# B&R Automation Studio project dbserv_0640 (part 13)

#### iec60870_5_103.c
```c
#ifdef _DEFAULT_INCLUDES
	#include <AsDefault.h>
#endif
/******************************************************************************
*    COPYRIGHT    BERNECKER + RAINER Industrie-Elektronik Ges.m.b.H           *
*******************************************************************************
*  Projekt:  Protokoll Treiber IEC 60870-5-103
*  Teil:     Hauptprogramm
*  Datei:    iec60870_5_103.c
*  Typ:      GNU-C (32 Bit)
*------------------------------------------------------------------------------
*  Revision: 03.00.5
*  Datum:    07-02-2019
*  Autor:    KOB
*------------------------------------------------------------------------------
*  Funktion:
*------------------------------------------------------------------------------
*  Rev.   | Datum    | Name | Kommentar
*  -------+----------+------+---------------------------------------------------
*  01.00  | 26-11-03 | KOB  | Datei-Erstellung
*  01.01  | 09-02-04 | KOB  | Debugkonfiguration um Liniennummer erweitert
*         |          |      | Meldung an LS, falls Schnittstelle nicht geöffnet werden
*		  |          |      | kann, dabei warten bis myidBrServer!= 0 ist.
*  01.02  | 07-05-04 | KOB  | Verbindungsstoerung bei Initialisierung auf 1 setzen, damit
*		  |          |      | beim ersten gültigen Telegramm der Datenpunkt Kopplungsstoerung
*		  |          |      | beschrieben wird.
*  01.03  | 15-12-04 | KOB  | Bei ungültigen Analogwerten (Invalid oder Overflow) wird
*         |          |      | als Ersatzwert 7FFF gesendet.
*  01.04  | 11-04-06 | WAI  | FileIO-Library includiert wegen neuer dbServ-Version mit Archivierung
*  01.05  | 24-05-06 | KOB  | Telegrammauswertung flexibler gestaltet (wegen anderem Verhalten von ABB)
*		  |          |      |
*  01.06  | 10-01-07 | KOB  | Erweiterung um die Telegramme:
*         |          |      | Type Identification 3 : Measurands 1
*         |          |      | (check_m3, iec__103_sub.c)
*         |          |      | Type Identification 79: Privates Telegramm zur Übertragung von Zählwerten
*         |          |      | (check_m79, iec__103_sub.c)
*         |          |      | Auswertung der im privaten Telegramm empfangenen Zählwerte
*         |          |      | (save_analogwert_priv, iec__103_serv.c)
*		  |          |      |
*  02.05.1| 02-09-08 | KOB  | Neue Modi für Doppelmeldungen:
*		  |			 |		| DOPPEL_EINZEL_NORMAL_NOINVALID und DOPPEL_EINZEL_INVERS_NOINVALID
*		  |          |      |
*		  |			 |		| KE_Init: Bei der Auswertungt des Rückmeldetelegrammes
*		  |			 |		| Identification Message (check_m5) wird die Überprüfung des
*		  |			 |		| Function Type weggelassen, d.h. es wird für alle Geräte aktzeptiert.
*		  |			 |		| Bisher wurde das Telegramm nur für Function Type 160,192,240 zugelassen.
*		  |          |      |
*         |          |      |
*  02.05.2| 02-09-08 | KOB  | Funktionen wie unter 01.06 beschrieben eingefügt.
*         |          |      |
*  02.06.4| 27-09-10 | WAI  | IsANumber() mit Vorzeichen
*         |          |      |
*  02.07.2| 26-07-11 | KOB  | Erweiterung um die Telegramme:
*         |          |      | Type Identification 205: Privates Telegramm zur Übertragung von Zählwerten (Siemens)
*         |          |      | (check_m205, iec__103_sub.c)
*         |          |      | Auswertung der im privaten Telegramm empfangenen Zählwerte
*         |          |      | (save_counter_2, iec__103_serv.c)
*         |          |      |
* 		  |			 | KOB  | Ueberwachung der Zeitsynchronisation:
*         |          |      | Parameter IEC Global: Timeout fuer Rueckmeldung Zeitsyncronisation (TIME.TIMEOUT)
*         |          |      | Parameter pro Gerät : ERR.TIMESYNC
*  02.07.3| 04-12-13 | KOB  | check_m5 angepasst: Zustand von ACD Bit ignoriert, Kompatibilitätsmodus 3 akzeptieren
*         |          |      | check_m6 angepasst: nicht verwendete Bits der zurueckgemeldeten Zeit ausmaskieren
*         |          |      | neue Debug Möglichkeit (Variablen: IEC_Info_Clear,IEC_Info_Enable,IEC_InfoNumber,IEC_Info)
*         |          |      | Aufschlüsselung der IEC Telegrammsteuerelemente und Eintrag in Buffer
*  03.00.2| 28-01-14 | KOB  | check_m5 angepasst: Info Nr 2 akzeptieren
*         |          |      | Defaultwert für IEC_Config.TimeClass2PollFast von 100ms auf 200ms erhöht
*  03.00.3| 04-04-14 | KOB  | TIME_DIFF_SYNCH_MAX von 2 auf 10 geändert
*         |          |      | DeviceActivType erweitert um die Elemente
*         |          |      | TDiff und TDiffCounter;
*         |          |      | check_m6() Uhrzeitdifferenz wird in Struktur eingetragen
*         |          |      | Ist die Uhrzeitdifferenz zu groß, wird erste beim 2.Mal Felhler generiert
*  03.00.4| 11-10-16 | WAI  | Änderungen tbd (BIE)
*  03.00.5| 07-02-19 | KOB  | Senden von Kommandos überarbeitet

******************************************************************************/

/***********************************************************************/
/* Headerfiles einbinden                                               */
/***********************************************************************/

#include <bur\plc.h>			/* RPS-spezifische Typendeklarationen */
#include <string.h>
#include <dvframe.h>
#include <asbrstr.h>
#include <sys_lib.h>
#include <brsystem.h>
#include <fileio.h>
#include "iec__103_date.h"		/* Funktionen zur Datumsberechnung */
#include "iec60870_5_103.h"		/* Definition der globalen Variablen */
#include "iec__103_debug.h"		/* Funktionen fuer Ausgabe von Debug-Meldungen */
#include "iec__103_parse.h"		/* Parser Funktionen */
#include "dbserv.h"				/* Meldeserver */

extern DebugConfig_typ	DebugConfig;

/***********************************************************************/
/* 					Initialisierungs-Unterprogramm                     */
/***********************************************************************/

void _INIT init_iec(void)
{
	signed short i,n;

	/*--------------------------------*/
	/* Variablen initialisieren       */
	/*--------------------------------*/
	for(i=0;i<ITEM_DIAGNOSE_SIZE;i++) {
		IEC_ItemDiagnose[i].showData	= 0;
	}
	IEC_NormDiagnose.showData			= 0;

	dbg_buf_iec_clear();
	IEC_Info_Clear	= 0;
	IEC_Info_Enable = 0;

	memset(&SYS_Statistic,0,sizeof(SYS_Statistic));
	memset(&DistDataServer,0,sizeof(DistDataServer));						/* Variable fuer die Uebergabe von Stoerschrieben an das Leitsystem */
	memset(&stANL,0,sizeof(stANL));											/* Variable für Linien und Geräteverwaltung */
	memset(&stComIni,0,sizeof(stComIni));									/* Variable zur Verwaltung der Schnittstellen */

	myidBrServer			= 0;											/* ID BR-Server */
	DisturbanceSimulation	= 0;											/* Merker zur Simulation eines Stoerschriebes */

	rt_info.enable = 1; 													/* Taskklassenzykluszeit ermitteln */
	RTInfo(&rt_info);
	if(rt_info.status==0)	CycleTime	= (rt_info.cycle_time / 1000);		/* Zykluszeit in ms */
	else 					CycleTime	= 10;								/* Zykluszeit in ms */

	DebugConfig.OpenDevice			= 0;									/* Debug Funktion deaktivieren */
	DebugConfig.DebugEnable			= 0;
	DebugConfig.DebugDelayAdresse	= 0;
	DebugConfig.DebugDelayTime		= 0;
	DebugConfig.DebugDelayCounter	= 0;

	Error	= 0;															/* Generelle Variable fuer Initialisierungsfehler */

	/*----------------------------------------------------------------------*/
	/* initialize debugging 												*/
	/*----------------------------------------------------------------------*/

	#ifdef DEBUG
		debug_initialize();
	#endif

	/*--------------------------------------------------*/
	/* Globale Konfigurationsparameter initialisieren	*/
	/*--------------------------------------------------*/

	IEC_Config.TimeOut				= 100;				/* Timeout bei Telegrammempfang (in ms) */
	IEC_Config.RetryAnz				= 6;				/* Anzahl Telegrammwiederholungen bei bestehender Verbindung */
	IEC_Config.ConnAnz				= 3;				/* Anzahl Telegrammwiederholung bei neu aufzubauender Verbindung */
	IEC_Config.WaitIntv				= 100000;			/* Wartezeit für erneuten Verbindungsaufbau (in ms) */
	IEC_Config.TimeTS				= 60000;			/* Intervallzeit fuer Uhrzeitsynchronisation (in ms) */
	IEC_Config.TimeOutTimeSynch		= 10000;			/* Timeout fuer die Rückantwort bei Zeitsynchronisation in (ms) */
	IEC_Config.EnableComReset		= 1;				/* Freigabe fuer das Schliessen und Wieder-Oeffnen der Schnittstelle bei Schreibfehlern */
	IEC_Config.TimeClass2Poll		= 1000;				/* Abtastzeit Class 2 Telegramme (Analogwerte) (in ms) */
	IEC_Config.TimeClass2PollFast	= 200;				/* Abtastzeit Class 2 Telegramme (Analogwerte) (in ms) während Übertragung von Störschrieben in ms */
	IEC_Config.DistDataTimeoutMax	= 20000;			/* Timeout fuer den Telegrammempfang bei Stoerschriebuebertragung in (ms) */
	IEC_Config.DistDataEnable		= 1;				/* Freigabe fuer Stoerschriebuebertragung */
	IEC_Config.DisturbanceDelay		= 10000;			/* Zeit die ein Lesen von Stoerschrieben der gleichen Station verzoegert wird in (ms) */
	IEC_Config.CommandEnable		= 0;				/* Freigabe für die Übertragung von Kommandos */
	IEC_Config.CommandTimeoutMax	= 40000;			/* Timeout fuer die Uebertragung von Kommandos in (ms) */

	/*****************************************************************************/
	/* Initialisierung nach Konfigurationsdatenmodul dplist und typlist (DbServ) */
	/*****************************************************************************/
#ifdef INIT_MODE_DM_DPLIST

	/*--------------------------------------------------*/
	/* Konfiguration aus Konfigurationsmodulen auslesen */
	/*--------------------------------------------------*/

	for(aktANL= 0; aktANL < MAX_LINES; aktANL++) {
		for(n = 0; n < DEVICES_PRO_LINE; n++) {
			stANL[aktANL].DeviceActiv[n].FaultFunctionType		= 160; /* Vorbelegung, wird später vom Telegramm des Geräts übernommen */
		}
	}

	iec_parser();

	Error = IEC_ParserInfo.error;

	/* Kein Schwerwiegender Fehler beim Parsen */
	if(Error==0) {
		/* Maximale Anzahl Linien (Endevariable für Schleifen) */
		if(IEC_ParserInfo.NrOfLines>0) {
			maxANL = IEC_ParserInfo.NrOfLines - 1;
		}
		else {
			maxANL = 0;
		}

		for(aktANL= 0; aktANL <= maxANL; aktANL++) {
			stANL[aktANL].LinienNummer			= IEC_GlobalData.Line[aktANL].LineNr.value;
			stANL[aktANL].Error					= IEC_ParserInfo.Line[aktANL].error;
			stANL[aktANL].dm.AdrDM_norm			= IEC_ParserInfo.memAdr;
			stANL[aktANL].dm.MaxWerteDM_norm	= IEC_ParserInfo.NrOfNormValues;
			stANL[aktANL].dm.AdrDM_wert			= IEC_ParserInfo.Line[aktANL].memAdr;
			stANL[aktANL].dm.MaxWerteDM_wert	= IEC_ParserInfo.Line[aktANL].NrOfItems;

			stANL[aktANL].DeviceAtWork 			= 0;
			for(n = 0; n < DEVICES_PRO_LINE; n++) {
				stANL[aktANL].DeviceActiv[n].Enabled = stANL[aktANL].DeviceTAB[n].Aktiv;
				if(stANL[aktANL].DeviceActiv[n].Enabled) {
					stANL[aktANL].DeviceActiv[n].Adresse 				= stANL[aktANL].DeviceTAB[n].Adresse;
					stANL[aktANL].DeviceActiv[n].AdresseLeitsystem 		= 1;
					stANL[aktANL].DeviceActiv[n].AnlagenNr				= stANL[aktANL].DeviceTAB[n].AnlagenNr;
					stANL[aktANL].DeviceActiv[n].Verbindungsversuche	= 0;
					stANL[aktANL].DeviceActiv[n].VerbindungsStoerung	= 1;	/* Sorgt fuer Eintrag in Datenbank bei bestehender Verbindung */
					stANL[aktANL].DeviceActiv[n].ZeitLetzteVerbindung	= 0;
					stANL[aktANL].DeviceActiv[n].ZeitsynchAktiv			= 0;
					stANL[aktANL].DeviceActiv[n].StateTimeSynchError	= STATE_ERROR_UNDEFINED;
					stANL[aktANL].DeviceActiv[n].TimeoutTimeSynch		= 0;
					stANL[aktANL].DeviceActiv[n].FCB_Toggle				= 0;
					stANL[aktANL].DeviceActiv[n].KE_InitOk				= 0;
					stANL[aktANL].DeviceActiv[n].ZeitLetzteZeitsync		= IEC_Config.TimeTS;
					stANL[aktANL].DeviceActiv[n].Class1Request			= 0;
					stANL[aktANL].DeviceActiv[n].TimoutNext				= 0;
					stANL[aktANL].DeviceActiv[n].GI_Ok					= 0;
					stANL[aktANL].DeviceActiv[n].LetzterACD				= 0;
					stANL[aktANL].DeviceActiv[n].Class2Verz				= 0;
					stANL[aktANL].DeviceActiv[n].Class1Verz				= 0;
				}
				if(stANL[aktANL].DeviceActiv[n].Enabled && !stANL[aktANL].DeviceAtWork) {
					stANL[aktANL].DeviceAtWork = n + 1;
				}
			}
		}
	}
#endif

	/*****************************************************************************/
	/* Initialisierung mit Datenmoduln lines,devax,wertx,mruc,norm               */
	/*****************************************************************************/
#ifdef INIT_MODE_DM_WERT

	/*----------------------------------------------------------------------*/
	/* read data-modul lines 												*/
	/*----------------------------------------------------------------------*/

	DOI_lines.enable	= 1;
	DOI_lines.pName	= (UDINT) "lines";

	DatObjInfo(&DOI_lines);

	if(DOI_lines.status==0) {
		DOR_lines.enable 		= 1;
		DOR_lines.ident 		= DOI_lines.ident;
		DOR_lines.Offset 		= 0;
		DOR_lines.len			= sizeof(ActiveLines);
		DOR_lines.pDestination	= (UDINT) &ActiveLines;
		DatObjRead(&DOR_lines);

		if(ActiveLines>MAX_LINES) ActiveLines = MAX_LINES;

		if(ActiveLines>0)		maxANL = ActiveLines - 1;
		else					maxANL = 0;

		DOR_lines.Offset 		= 2;
		DOR_lines.enable 		= 1;
		DOR_lines.ident 		= DOI_lines.ident;
		for(aktANL = 0; aktANL <= maxANL; aktANL++) {
			DOR_lines.len			= sizeof(stANL[aktANL].LinienNummer);
			DOR_lines.pDestination	= (UDINT) &stANL[aktANL].LinienNummer;
			DatObjRead(&DOR_lines);
			DOR_lines.Offset 		+= 2;
		}

		DOR_lines.Offset 		= 14;
		DOR_lines.enable 		= 1;
		DOR_lines.ident 		= DOI_lines.ident;
		DOR_lines.len			= sizeof(DistDataType);
		DOR_lines.pDestination	= (UDINT) &DistDataType;
		DatObjRead(&DOR_lines);

		DOR_lines.Offset 		+= 2;
		DOR_lines.enable 		= 1;
		DOR_lines.ident 		= DOI_lines.ident;
		DOR_lines.len			= sizeof(DistDataPoint);
		DOR_lines.pDestination	= (UDINT) &DistDataPoint;
		DatObjRead(&DOR_lines);

		DOR_lines.Offset 		= 20;
		for(aktANL = 0; aktANL <= maxANL; aktANL++) {
			DOR_lines.len			= 23;
			DOR_lines.pDestination	= (UDINT) &stComIni[aktANL].StringDevice;
			DatObjRead(&DOR_lines);
			DOR_lines.Offset 		+= 24;

			DOR_lines.len			= 79;
			DOR_lines.pDestination	= (UDINT) &stComIni[aktANL].StringMode;
			DatObjRead(&DOR_lines);
			DOR_lines.Offset 		+= 80;

			for(i=sizeof(stComIni[aktANL].StringDevice)-1; i>=0;i--) {
				if((stComIni[aktANL].StringDevice[i]!=' ') && (stComIni[aktANL].StringDevice[i]!=0)) break;
				if(stComIni[aktANL].StringDevice[i]==' ') stComIni[aktANL].StringDevice[i] = 0;
			}
			for(i=sizeof(stComIni[aktANL].StringMode)-1; i>=0;i--) {
				if((stComIni[aktANL].StringMode[i]!=' ') && (stComIni[aktANL].StringMode[i]!=0)) break;
				if(stComIni[aktANL].StringMode[i]==' ') stComIni[aktANL].StringMode[i] = 0;
			}
		}
	}
	else {
		Error	= INI_ERR_DO_LINES;
		maxANL	= 0;
	}

	/*----------------------------------------------------------------------*/
	/* read data-modul mruk 												*/
	/*----------------------------------------------------------------------*/

	DOI_mruk.enable	= 1;
	DOI_mruk.pName	= (UDINT) "mruk";

	DatObjInfo(&DOI_mruk);

	if(DOI_mruk.status==0) {
		for(aktANL=0; aktANL<=maxANL; aktANL++) {
			stANL[aktANL].dm.AdrDM_mruk			= DOI_mruk.pDatObjMem;
			stANL[aktANL].dm.MaxWerteDM_mruk	= DOI_mruk.len / 2;
		}
	}
	else {
		for(aktANL=0; aktANL<=maxANL; aktANL++) {
			stANL[aktANL].dm.AdrDM_mruk			= 0;
			stANL[aktANL].dm.MaxWerteDM_mruk	= 0;
		}
		Error = INI_ERR_DO_MRUK;
	}

	/*----------------------------------------------------------------------*/
	/* read data-modul norm 												*/
	/*----------------------------------------------------------------------*/

	DOI_norm.enable	= 1;
	DOI_norm.pName	= (UDINT) "norm";

	DatObjInfo(&DOI_norm);

	if(DOI_norm.status==0) {
		for(aktANL=0; aktANL<=maxANL; aktANL++) {
			stANL[aktANL].dm.AdrDM_norm			= DOI_norm.pDatObjMem;
			stANL[aktANL].dm.MaxWerteDM_norm	= DOI_norm.len / 8;
		}
	}
	else {
		for(aktANL=0; aktANL<=maxANL; aktANL++) {
			stANL[aktANL].dm.AdrDM_norm			= 0;
			stANL[aktANL].dm.MaxWerteDM_norm	= 0;
		}
		Error = INI_ERR_DO_NORM;
	}

	/*----------------------------------------------------------------------*/
	/* read data-modul deva and wert for line 1 to n											*/
	/*----------------------------------------------------------------------*/

	for(aktANL=0; aktANL<=maxANL; aktANL++) {
		if(!stANL[aktANL].Error) {
			DOI_deva[aktANL].enable	= 1;
			switch(aktANL) {
				case 0:	DOI_deva[aktANL].pName	= (UDINT) "deva1"; break;
				case 1:	DOI_deva[aktANL].pName	= (UDINT) "deva2"; break;
				case 2:	DOI_deva[aktANL].pName	= (UDINT) "deva3"; break;
				case 3:	DOI_deva[aktANL].pName	= (UDINT) "deva4"; break;
				case 4:	DOI_deva[aktANL].pName	= (UDINT) "deva5"; break;
				case 5:	DOI_deva[aktANL].pName	= (UDINT) "deva6"; break;
			}

			DatObjInfo(&DOI_deva[aktANL]);

			if(DOI_deva[aktANL].status!=0) {
				stANL[aktANL].Error = INI_ERR_DO_DEVA;
			}
			else {
				if(DOI_deva[aktANL].len>sizeof(stANL[aktANL].DeviceTAB)) {
					DOR_deva[aktANL].len = sizeof(stANL[aktANL].DeviceTAB);
				}
				else {
					DOR_deva[aktANL].len = DOI_deva[aktANL].len;
				}

				DOR_deva[aktANL].enable 		= 1;
				DOR_deva[aktANL].ident 			= DOI_deva[aktANL].ident;
				DOR_deva[aktANL].Offset 		= 0;
				DOR_deva[aktANL].pDestination	= (UDINT) &stANL[aktANL].DeviceTAB;

				DatObjRead(&DOR_deva[aktANL]);

				if(DOR_deva[aktANL].status != 0) {
					stANL[aktANL].Error = INI_ERR_DO_DEVA_READ;
				}
				else {
					stANL[aktANL].DeviceAtWork = 0;
					for(n = 0; n < DEVICES_PRO_LINE; n++) {
						stANL[aktANL].DeviceActiv[n].Enabled = stANL[aktANL].DeviceTAB[n].Aktiv;
						if(stANL[aktANL].DeviceActiv[n].Enabled) {
							stANL[aktANL].DeviceActiv[n].Adresse 				= stANL[aktANL].DeviceTAB[n].Adresse;
							stANL[aktANL].DeviceActiv[n].AdresseLeitsystem 		= stANL[aktANL].LinienNummer + stANL[aktANL].DeviceTAB[n].Adresse;
							stANL[aktANL].DeviceActiv[n].AnlagenNr				= stANL[aktANL].DeviceTAB[n].AnlagenNr;
							stANL[aktANL].DeviceActiv[n].Verbindungsversuche	= 0;
							stANL[aktANL].DeviceActiv[n].VerbindungsStoerung	= 1;
							stANL[aktANL].DeviceActiv[n].ZeitLetzteVerbindung	= 0;
							stANL[aktANL].DeviceActiv[n].ZeitsynchAktiv			= 0;
							stANL[aktANL].DeviceActiv[n].FCB_Toggle				= 0;
							stANL[aktANL].DeviceActiv[n].KE_InitOk				= 0;
							stANL[aktANL].DeviceActiv[n].ZeitLetzteZeitsync		= IEC_Config.TimeTS;
							stANL[aktANL].DeviceActiv[n].Class1Request			= 0;
							stANL[aktANL].DeviceActiv[n].TimoutNext				= 0;
							stANL[aktANL].DeviceActiv[n].GI_Ok					= 0;
							stANL[aktANL].DeviceActiv[n].LetzterACD				= 0;
							stANL[aktANL].DeviceActiv[n].Class2Verz				= 0;
							stANL[aktANL].DeviceActiv[n].Class1Verz				= 0;
							stANL[aktANL].DeviceActiv[n].FaultFunctionType		= 160; /* Vorbelegung, wird später vom Telegramm des Geräts übernommen */
						}
						if(stANL[aktANL].DeviceActiv[n].Enabled && !stANL[aktANL].DeviceAtWork)
							stANL[aktANL].DeviceAtWork = n + 1;
					}
				} /* if(DOR_deva[aktANL].status != 0)  */
			} /* if(DOI_deva[aktANL].status!=0)  */
		} /* if(!stANL[aktANL].Error) */

		if(!stANL[aktANL].Error) {
			DOI_wert[aktANL].enable	= 1;
			switch(aktANL) {
				case 0:	DOI_wert[aktANL].pName	= (UDINT) "wert1"; break;
				case 1:	DOI_wert[aktANL].pName	= (UDINT) "wert2"; break;
				case 2:	DOI_wert[aktANL].pName	= (UDINT) "wert3"; break;
				case 3:	DOI_wert[aktANL].pName	= (UDINT) "wert4"; break;
				case 4:	DOI_wert[aktANL].pName	= (UDINT) "wert5"; break;
				case 5:	DOI_wert[aktANL].pName	= (UDINT) "wert6"; break;
			}

			DatObjInfo(&DOI_wert[aktANL]);

			if(DOI_wert[aktANL].status==0) {
				stANL[aktANL].dm.AdrDM_wert			= DOI_wert[aktANL].pDatObjMem;
				stANL[aktANL].dm.MaxWerteDM_wert	= DOI_wert[aktANL].len / 8;
			}
			else {
				stANL[aktANL].Error = INI_ERR_DO_WERT;
			}
		}

	} /* for(aktANL=0; aktANL<=maxANL; aktANL++) */

#endif

	/*-----------------------------------------------------------------------------------*/
	/* Struktur zur Verwaltung der Linien und Geräte mit Konfigurationsdaten beschreiben */
	/*-----------------------------------------------------------------------------------*/

	for(aktANL = 0; aktANL <= MAX_LINES-1; aktANL++) {
		stANL[aktANL].com.receive_timeout	= IEC_Config.TimeOut;	/* Timeout für Empfangstelegramm in ms */
		stANL[aktANL].com.Ident 			= 0;
		stANL[aktANL].com.OpenError			= 0;
		stANL[aktANL].com.WriteError		= 0;
		stANL[aktANL].com.WriteErrorCount	= 0;
		stANL[aktANL].com.FirstWriteError	= 0;
		stANL[aktANL].com.ReOpenCount		= 0;
		stANL[aktANL].ComStart				= 1;					/* Freigabe für Kommunikation */
		stANL[aktANL].DistData.Function		= NO_FUNCTION;
		stANL[aktANL].DistData.DataSend		= 0;
		stANL[aktANL].Command.Function		= NO_FUNCTION;
		stANL[aktANL].SNr					= 0;
	}

	/*----------------------------------------------------------------------*/
	/* initialize and open interface for line 1 to n						*/
	/*----------------------------------------------------------------------*/

	/* initialize config structure */

	for(aktANL=0; aktANL<=maxANL; aktANL++) {
		if(!stANL[aktANL].Error) {
			stComIni[aktANL].XOpenConfigStruct.idle		= 4;
			stComIni[aktANL].XOpenConfigStruct.delimc	= 0;
			stComIni[aktANL].XOpenConfigStruct.delim[0]	= 0;
			stComIni[aktANL].XOpenConfigStruct.delim[1]	= 0;
			stComIni[aktANL].XOpenConfigStruct.tx_cnt	= 2;
			stComIni[aktANL].XOpenConfigStruct.rx_cnt	= 2;
			stComIni[aktANL].XOpenConfigStruct.tx_len	= 256;
			stComIni[aktANL].XOpenConfigStruct.rx_len	= 256;
			stComIni[aktANL].XOpenConfigStruct.argc		= 0;
			stComIni[aktANL].XOpenConfigStruct.argv		= 0;

			/* initialize open structure */

			stComIni[aktANL].FrameXOpenStruct.device	= (UDINT) stComIni[aktANL].StringDevice;
			stComIni[aktANL].FrameXOpenStruct.mode		= (UDINT) stComIni[aktANL].StringMode;
			stComIni[aktANL].FrameXOpenStruct.config	= (UDINT) &stComIni[aktANL].XOpenConfigStruct;
			stComIni[aktANL].FrameXOpenStruct.enable	= 1;

			/* open interface */

			FRM_xopen(&stComIni[aktANL].FrameXOpenStruct); 						/* open an interface */
			if (stComIni[aktANL].FrameXOpenStruct.status != 0) {				/* check status */
				stANL[aktANL].com.OpenError = 1;
				stANL[aktANL].Error			= INI_ERR_DEVICE_OPEN;
				strcpy(MsgTxt,"Fehler beim Oeffnen von: ");
				strcat(MsgTxt,stComIni[aktANL].StringDevice);
				ErrStatistics("iec103", ERRLOG, stANL[aktANL].Error, stComIni[aktANL].FrameXOpenStruct.status, ERR_MSG_PRE_STRG, MsgTxt);
			}
			else {
				stANL[aktANL].com.Ident = stComIni[aktANL].FrameXOpenStruct.ident; 	/* get ident */
			}
		}
	}

	/*-------------------------------*/
	/* Buffer fuer Stoerschriebdaten */
	/*-------------------------------*/

	memset(&DataBuffer,0,sizeof(DataBuffer));

	if(IEC_Config.DistDataEnable) {								/* Freigabe fuer Stoerschriebuebertragung */

		/* Speicher fuer die Buffer allokieren */

		for(i=0;i<NR_OF_BUFFERS;i++) {
			DataBuffer.Info[i].Size = BUFFER_SIZE;
			DataBuffer.Info[i].status = TMP_alloc(DataBuffer.Info[i].Size, (void**)&DataBuffer.Info[i].DataAdr); 	/* allocate new memory from RAM*/
			if(DataBuffer.Info[i].status==0) {
				DataBuffer.NrOfBuffers++;
			}
			else {
				strcpy(MsgTxt,"Fehler TMP_alloc Stoerschrieb");
				ErrStatistics("iec103", ERRLOG, 0, DataBuffer.Info[i].status, ERR_MSG_PRE_STRG, MsgTxt);
			}
		}
	}

	/*-------------------------------*/
	/* Startschritt bestimmen        */
	/*-------------------------------*/

	for(aktANL=0; aktANL<=maxANL; aktANL++) {
		if(!stANL[aktANL].ComStart) {
			stANL[aktANL].SNr = 4;
		}
		else {
			if(stANL[aktANL].Error) {
				stANL[aktANL].SNr = 3;
			}
			else {
				stANL[aktANL].SNr = 0;
			}
		}
	}
}

/***********************************************************************/
/* 						zyklisches Hauptprogramm                       */
/***********************************************************************/

void _CYCLIC cyclic_iec(void)
{

	plcbit	found;
	UINT error,i,n;
	UINT LineIdx=0;
	UINT DeviceIdx=0;
	RTCtime_typ SysTime;
	DeviceActivType *pDeviceActiv;

	pDeviceActiv = &(stANL[0].DeviceActiv[0]);		/* nur um Compiler-Warnung zu verhindern */

	/* Einlesen der Echtzeituhr */

    error = RTC_gettime(&SysTime);
    if(error==0) {
      memcpy(&RPSTime,&SysTime,sizeof(RPSTime));
      RPSTimeOK = 1;
	}

	/* ID Meldeserver besorgen */

	get_idBrServer();

	/* Pruefen, ob Stoerschriebe angefordert bzw. geloeschet werden muessen */

	check_dist_data_transmission();

	/* Testfunktion für Onlinemonitor */

	if(DigTest.enable==1)
	{
		DigTest.enable	= 0;
		DigTest.ready	= 0;

		/* Liniennummer vorhanden ? */
		found = 0;
		for(n = 0; n <= maxANL; n++) {
			if(stANL[n].LinienNummer == DigTest.LinienNummer) {
				found	= 1;
				LineIdx	= n;
			}
		}

		/* Geraeteadresse vorhanden ? */
		if(found) {
			found = 0;
			for(n = 0; n < DEVICES_PRO_LINE; n++) {
				if(stANL[LineIdx].DeviceActiv[n].Adresse == DigTest.DeviceAdresse) {
					found		= 1;
					DeviceIdx	= n;
				}
			}
		}

		if(found) {
			save_digitalwert(	(DMInfoType *) &stANL[LineIdx].dm,
								stANL[LineIdx].LinienNummer,
								(DeviceActivType *) &stANL[LineIdx].DeviceActiv[DeviceIdx],
								DigTest.FunctionType,
								DigTest.InformationNumber,
								DigTest.Messwert,
								&RPSTime,
								stANL[LineIdx].DeviceActiv[0].set_event);						/* Event für Leitsystem */
			DigTest.ready	= 1;
		}
	}

	if(AnaTest.enable==1)
	{
		AnaTest.enable	= 0;
		AnaTest.ready	= 0;

		/* Liniennummer vorhanden ? */
		found = 0;
		for(n = 0; n <= maxANL; n++) {
			if(stANL[n].LinienNummer == AnaTest.LinienNummer) {
				found	= 1;
				LineIdx	= n;
			}
		}

		/* Geraeteadresse vorhanden ? */
		if(found) {
			found = 0;
			for(n = 0; n < DEVICES_PRO_LINE; n++) {
				if(stANL[LineIdx].DeviceActiv[n].Adresse == AnaTest.DeviceAdresse) {
					found		= 1;
					DeviceIdx	= n;
				}
			}
		}

		if(found) {
			save_analogwert	(	(DMInfoType *) &stANL[LineIdx].dm,
								stANL[LineIdx].LinienNummer,
								(DeviceActivType *) &stANL[LineIdx].DeviceActiv[DeviceIdx],
								AnaTest.FunctionType,
								AnaTest.InformationNumber,
								AnaTest.AnzahlMesswerte,
								(USINT *) &AnaTest.Messwerte,
     							stANL[LineIdx].DeviceActiv[0].set_event);						/* Event für Leitsystem */
			AnaTest.ready	= 1;
		}
	}

	if(GlobalTest.enable==1)
	{
		GlobalTest.enable = 0;
/*		set_global_event_station (idMessageServer, RPSTime, (UINT) GlobalTest.Adresse);*/
	}

	/* Uebergabe von Stoerschriebdaten aus einem Datenmodul an den Meldeserver */
	disturbance_simulation();

	iec_mem_diagnose();

	// Hilfsbuffer fuer IEC Diagnose
	if(IEC_Info_Clear) {
		dbg_buf_iec_clear();
		IEC_Info_Clear = 0;
	}

	/* Bis hierher nur Test */

	#ifdef DEBUG
		debug_open_device(DebugConfig.OpenDevice);
	#endif

	if ((Error == 0) && (myidBrServer!=0)) {

		for(aktANL=0; aktANL<=maxANL; aktANL++) {

				switch(stANL[aktANL].SNr) {
					case 0:		/* Normaler Schreib- Lesebetrieb */
						Zeitmessung(&stANL[aktANL]);
						Device_Reaktivieren(&stANL[aktANL]);
						disturbance_data_timeout(&stANL[aktANL]);
						command_timeout(&stANL[aktANL]);
						timesynch_timeout(&stANL[aktANL]);

						if(stANL[aktANL].com.write_read_activ == WRITE) {
							Data_write(&stANL[aktANL]);
						}
						else {
							Data_read(&stANL[aktANL]);
						}

						FrameReadStruct.enable = 1;
						FrameReadStruct.ident = stANL[aktANL].com.Ident;

						FRM_read(&FrameReadStruct); 								/* read data form interface */

						ReadBuffer 			= (UDINT*) FrameReadStruct.buffer;		/* get adress of read buffer */
						ReadBufferLength	= FrameReadStruct.buflng; 				/* get length of read buffer */
						StatusRead			= FrameReadStruct.status; 				/* get status */

						if (StatusRead == 0) {										/* check status */
							if((ReadBufferLength + stANL[aktANL].com.RBufferAdr)<=sizeof(stANL[aktANL].com.ReadData)) {
								memcpy(&stANL[aktANL].com.ReadData[stANL[aktANL].com.RBufferAdr], ReadBuffer, ReadBufferLength);/* copy read data into array */
						 		stANL[aktANL].com.RBufferAdr += ReadBufferLength;
							}

							if(stANL[aktANL].DeviceAtWork>0)
								pDeviceActiv = &(stANL[aktANL].DeviceActiv[stANL[aktANL].DeviceAtWork-1]);

							#ifdef DEBUG
								dbg_msg(READBUFFER,
										stANL[aktANL].com.RBufferAdr,
										0,
										stANL[aktANL].LinienNummer,
										pDeviceActiv->Adresse,
										0,
										0,
										0,
										stANL[aktANL].com.ReadData);
							#endif
																					/* initialize release buffer structure */
							FrameReleaseBufferStruct.enable = 1;
							FrameReleaseBufferStruct.ident = stANL[aktANL].com.Ident;
							FrameReleaseBufferStruct.buffer = (UDINT) ReadBuffer;
							FrameReleaseBufferStruct.buflng = ReadBufferLength;

							FRM_rbuf(&FrameReleaseBufferStruct); 						/* release read buffer */

							StatusReleaseBuffer = FrameReleaseBufferStruct.status; 		/* get status */

							if (StatusReleaseBuffer != 0)  								/* check status */
								ReadError = 1; 											/* set error level for FRM_rbuf */
						}
						if((stANL[aktANL].com.WriteErrorCount>3) && (IEC_Config.EnableComReset)) stANL[aktANL].SNr++;
						break;

					case 1:		/* Schnittstelle schliessen */
						/* initialize close structure */
						FrameCloseStruct.ident	= stANL[aktANL].com.Ident;
						FrameCloseStruct.enable = 1;
						FRM_close(&FrameCloseStruct); 					/* close interface */
						stANL[aktANL].SNr++;
						break;

					case 2:		/* Schnittstelle erneut oeffnen */
						FRM_xopen(&stComIni[aktANL].FrameXOpenStruct); 						/* open an interface */
						if (stComIni[aktANL].FrameXOpenStruct.status != 0) {				/* check status */
							stANL[aktANL].com.OpenError = 1;
							stANL[aktANL].Error			= INI_ERR_DEVICE_OPEN;
							stANL[aktANL].SNr			= 3;
						}
						else {
							stANL[aktANL].com.Ident				= stComIni[aktANL].FrameXOpenStruct.ident; 	/* get ident */
							stANL[aktANL].SNr 					= 0;
							stANL[aktANL].com.LastWriteError	= stANL[aktANL].com.WriteError;
							stANL[aktANL].com.WriteErrorCount	= 0;
							stANL[aktANL].com.WriteError		= 0;
						}

						stANL[aktANL].com.ReOpenCount++;
						break;

					/* Fehlermeldung aller Geräte: Verbindungsstoerung */
					case 3:
						if(myidBrServer!=0) {
							for(i=0;i<DEVICES_PRO_LINE;i++) {
								if(stANL[aktANL].DeviceTAB[i].Aktiv==0) continue;

								save_kopplungsstoerung( &(stANL[aktANL].dm),								/* Adresse Datenmodul-Infostruktur */
														stANL[aktANL].LinienNummer,							/* Liniennummer */
														(DeviceActivType *) &stANL[aktANL].DeviceActiv[i],
											 			2,													/* Messwert	(Doppelmeldung 1=aus 2=ein) */
							 							&RPSTime,											/* Zeitstempel 		 */
											 			TRUE);												/* Event für Leitsystem */
							}
							stANL[aktANL].SNr = 4;
						}
						break;

					/* Schritt 4: Keine Funktion */
					case 4:
						break;

				} /* switch */
		} /* for () */
	} /* if(Error==0) */
}

/*** eof *****************************************************************************/
```

#### iec60870_5_103.h
```c
/******************************************************************************
*    COPYRIGHT    BERNECKER + RAINER Industrie-Elektronik Ges.m.b.H           *
*******************************************************************************
*  Projekt:  Protokoll Treiber IEC 60870-5-103
*  Teil:     Hauptprogramm
*  Datei:    iec60870_5_103.h
*  Typ:      GNU-C (32 Bit)
*------------------------------------------------------------------------------
*  Revision: 03.00.4
*  Datum:    07-02-19
*  Autor:    KOB
*------------------------------------------------------------------------------
*  Funktion: Globale Headerdatei fuer IEC-Treiber
*------------------------------------------------------------------------------
*  Rev.   | Datum    | Name | Kommentar
*  -------+----------+------+---------------------------------------------------
*  01.00  | 26-11-03 | KOB  | Datei-Erstellung
*         |          |      |
*  01.06  | 10-01-07 | KOB  | Erweiterung um die Telegramme:
*         |          |      | Type Identification 3 : Measurands 1
*         |          |      | (check_m3, iec__103_sub.c)
*         |          |      | Type Identification 79: Privates Telegramm zur Übertragung von Zählwerten
*         |          |      | (check_m79, iec__103_sub.c)
*         |          |      | Auswertung der im privaten Telegramm empfangenen Zählwerte
*         |          |      | (save_analogwert_priv, iec__103_serv.c)
*         |          |      |
*  02.05.2| 02-09-08 | KOB  | Funktionen wie unter 01.06 beschrieben eingefügt.
*  02.05.2| 02-09-08 | KOB  | Funktionen wie unter 01.06 beschrieben eingefügt.
*  03.00.3| 04-04-14 | KOB  | TIME_DIFF_SYNCH_MAX von 2 auf 10 geändert
*         |          |      | DeviceActivType erweitert um die Elemente
*         |          |      | TDiff und TDiffCounter;
*  03.00.4| 07-02-19 | KOB  | Neue Konstante für Fehlermeldungen der Commando-Schreibfunktion
*         |          |      | Neuer Prototyp DeviceIsActive
******************************************************************************/
#include <bur/plctypes.h>
#include <dvframe.h>
#include <sys_lib.h>
#include <dataobj.h>
#include <brsystem.h>
#include <astime.h>
#include "bksys.h"

/***********************************************************************/
/* Konstantendefinition                                                */
/***********************************************************************/

/* ------------------------------ */
/* Quelle der Konfigurationsdaten */
/* ------------------------------ */

/* Je nach Definition werden die Konfigurationsdaten in den beschriebenen Datenmodulen erwartet */

/* Quelle der Konfigurationsdaten: dplist und typlist (DbServ) */
#define INIT_MODE_DM_DPLIST
/* Quelle der Konfigurationsdaten: lines,devax,wertx,mruc,norm (Ursprungsversion) */
#undef	INIT_MODE_DM_WERT

/* -------------------------------------------*/
/* Grenzwert fuer Linien und Geraete pro Linie */
/* -------------------------------------------*/

#define MAX_LINES							12				/* Maximal moegliche Anzahl Linien */
#define DEVICES_PRO_LINE					32				/* Anzahl moeglicher Geraete pro Linie */

/* -------------------------------------------*/
/* Buffer fuer Stoerschriebdaten			  */
/* -------------------------------------------*/

#define NR_OF_BUFFERS						6				/* Maximale Anzahl von Buffern fuer die Uebertragung von Stoerschrieben */
#define BUFFER_SIZE							150000			/* Groesse eines Buffers fuer die Uebertragung von Stoerschrieben */

#define MAX_ANALOGWERTE						16				/* Maximale Anzahl Analogwerte in einem Telegramm */
/* -------------------------------------------*/
/* Fehlerkennungen Initialisierung            */
/* -------------------------------------------*/

#define INI_ERR_DO_LINES					1				/* Fehler Datenmodul lines,   siehe: DOI_lines.status */
#define INI_ERR_DO_MRUK						2				/* Fehler Datenmodul mruk,    siehe: DOI_mruk.status	*/
#define INI_ERR_DO_NORM						3				/* Fehler Datenmodul norm,    siehe: DOI_norm.status	*/
#define INI_ERR_DEVICE_OPEN					100				/* Fehler Device Open,		  siehe: stComIni[].FrameXOpenStruct */
#define INI_ERR_DO_DEVA						103				/* Fehler Datenmodul deva_,   siehe: DOI_deva[].status */
#define INI_ERR_DO_DEVA_READ				104				/* Leseehler Datenmodul deva_,siehe: DOR_deva[].status */
#define INI_ERR_DO_WERT						105				/* Fehler Datenmodul wert_,   siehe: DOI_wert[].status */
#define INI_ERR_DO_STOER					106				/* Fehler Datenmodul stoer_,  siehe: DOI_stoer[].status */

/* -------------------------------------------*/
/* Fehlerkennungen Stoerschriebuebermittlung  */
/* -------------------------------------------*/

#define DIST_ERR_FAULTNUMBER				1001
#define DIST_ERR_TELEGRAM					1002
#define DIST_ERR_TRY_MAX_TAGS				1003
#define DIST_ERR_TRY_MAX_CHANNEL			1004
#define DIST_ERR_ABORT						1005
#define DIST_ERR_TAG_ABORT					1006
#define DIST_ERR_CHANNEL_ABORT				1007
#define DIST_ERR_TIMEOUT					1008
#define DIST_ERR_VAL_STARTPOS				1009
#define DIST_ERR_VAL_ENDPOS					1010
#define DIST_ERR_NR_OF_CHANNELS				1011
#define DIST_ERR_CHANNEL_TYPE				1012
#define DIST_ERR_MEMORY						1013
#define DIST_ERR_LINK_DOWN					1014
#define DIST_ERR_RECEIVE_ERROR				1015

/* -------------------------------------------*/
/* Fehlerkennungen fuer Kommandos             */
/* -------------------------------------------*/

#define COMMAND_ERR_TIMEOUT					2008
#define COMMAND_ERR_NAK						2020
#define COMMAND_ERR_FUNCTION_NR				2021
#define COMMAND_ERR_INFORMATION_NR			2022
#define COMMAND_ERR_VALUE					2023
#define COMMAND_ERR_RETURNINFORMATION		2024
#define COMMAND_ERR_DISABLED				2025
#define COMMAND_ERR_DEVICE_NOT_READY		2026
#define COMMAND_ERR_DEVICE_ADR				2027
#define COMMAND_ERR_FUNCTION_ACTIVE			2028

/* --------------------------------------------*/
/* Allgemeine Konstanten                       */
/* --------------------------------------------*/

#define FALSE			0
#define TRUE			1

#define ACK				254
#define NAK				255

#define STATE_ERROR_UNDEFINED	0
#define STATE_ERROR_OFF			1
#define STATE_ERROR_ON			2

#define WRITE			0
#define READ			1

#define INIT_KE			1
#define INIT_KE_LAEUFT	2
#define ZEIT_SYNC		3
#define INIT_GI			4
#define INIT_GI_START   5
#define INIT_GI_LAEUFT	6
#define CLASS_1_REQ		7
#define CLASS_2_REQ		8
#define READY			99

#define TYPE_CONNECTION_ERROR	255		/* Typ für Datenpunkt : Verbindungsfehler */
#define INFO_CONNECTION_ERROR	255		/* Info für Datenpunkt: Verbindungsfehler */

#define TIME_DIFF_SYNCH_MAX		10		/* Erlaubte Zeitdifferenz nach Uhrzeitsynchronisation [s] */
/* -------------------------------------------------------------*/
/* Kennzeichnung für Einzelschritte der Störschriebübermittlung */
/* -------------------------------------------------------------*/

#define NO_FUNCTION							0
#define SELECTION_OF_FAULT	 				1
#define REQ_DISTURBANCE_TRANSMISSION		2
#define REQ_FOR_TAGS						3
#define REQ_FOR_A_CHANNEL					4
#define ACK_FOR_TAGS						5
#define ACK_FOR_A_CHANNEL					6
#define ACK_FOR_DISTURBANCE_DATA			7
#define REQ_FOR_LIST_OF_FAULTS				8
#define ABORT_DISTURBANCE_TRANSMISSION		9
#define ABORT_CHANNEL_TRANSMISSION			10

/* -------------------------------------------------------------------------*/
/* Kennung fuer Stoerschriebbuffer und Stoerschriebinformation des Geraetes */
/* -------------------------------------------------------------------------*/

#define NODATA								0
#define WRITE_BUFFER						1
#define DATA_READY							2
#define WAIT_FOR_QUIT						3
#define DELETE_DATA							4
#define SEND_DELETE_TELEGRAM				5
#define CLEAR_DATA_AGAIN					6

/* -------------------------------------------------------------------------*/
/* Kennzeichnung fuer das Speichern von Daten der Stoerschriebuebermittlung */
/* -------------------------------------------------------------------------*/

#define DISTURBANCE_START					1
#define DISTURBANCE_TAGS_START				2
#define DISTURBANCE_TAGS					3
#define DISTURBANCE_VALUES_START			4
#define DISTURBANCE_CHANNEL_START			5
#define DISTURBANCE_VALUES					6
#define DISTURBANCE_END						7

/* -------------------------------------------------------------------------*/
/* Befehlskennungen (Type of Order TOO) nach IEC 60870-5-103 7.2.6.26       */
/* -------------------------------------------------------------------------*/

#define DIST_DATA_TRANS_SUCCESSFULLY		64
#define DIST_DATA_TRANS_NOT_SUCCESSFULLY	65
#define ABORTION_OF_DIST_DATA				3
#define CHANNEL_TRANS_SUCCESSFULLY			66
#define CHANNEL_TRANS_NOT_SUCCESSFULLY		67
#define ABORTION_OF_CHANNEL					9
#define TAGS_TRANS_SUCCESSFULLY				68
#define TAGS_TRANS_NOT_SUCCESSFULLY			69
#define ABORTION_OF_TAGS					17

/* --------------------------------------------------------*/
/* Funktionskennungen bei der Uebertragung von Kommandos   */
/* --------------------------------------------------------*/

#define SEND_COMMAND						1
#define REPEAT_COMMAND						2
#define WAIT_FOR_COMMAND_ACK				3
#define WAIT_FOR_COMMAND_EXE				4

/***********************************************************************/
/* Datentypdeklaration                                                 */
/***********************************************************************/

/* ----------------------------------------*/
/* Konfigurationsvariable des IEC-Treibers */
/* ----------------------------------------*/
typedef struct
{
	unsigned long			TimeOut;					/* Timeout bei Telegrammempfang (in ms) */
	unsigned short			RetryAnz;					/* Anzahl Telegrammwiederholungen bei bestehender Verbindung */
	unsigned short			ConnAnz;					/* Anzahl Telegrammwiederholung bei neu aufzubauender Verbindung */
	unsigned long			WaitIntv;					/* Wartezeit für erneuten Verbindungsaufbau (in ms) */
	unsigned long			TimeTS;						/* Intervallzeit fuer Uhrzeitsynchronisation (in ms) */
	unsigned long			TimeOutTimeSynch;			/* Timeout fuer Rueckmeldetelegramm Zeitsynchronisation (ms) */
	unsigned short			EnableComReset;				/* Freigabe fuer das Schliessen und Wieder-Oeffnen der Schnittstelle bei Schreibfehlern */
	unsigned long			TimeClass2Poll;				/* Abtastzeit Class 2 Telegramme (Analogwerte) (in ms) */
	unsigned long			TimeClass2PollFast;			/* Abtastzeit Class 2 Telegramme (Analogwerte) während Übertragung von Störschrieben (in ms) */
	unsigned short			DistDataEnable;				/* Freigabe fuer Stoerschriebuebertragung */
	unsigned long			DistDataTimeoutMax;			/* Timeout fuer den Telegrammempfang bei Stoerschriebuebertragung in (ms) */
	unsigned long			DisturbanceDelay;			/* Zeit die ein Lesen von Stoerschrieben der gleichen Station verzoegert wird in (ms) */
	unsigned short			CommandEnable;				/* Freigabe fuer Kommandouebertragung */
	unsigned long			CommandTimeoutMax;			/* Timeout fuer die Uebertragung von Kommandos in (ms) */
} IEC_Config_typ;

/* Verwaltung der Unterstationen */

/*---------------------------------------------*/
/* Datenmodulstrukturen 		               */
/*---------------------------------------------*/

/*---------------------------------------------*/
/* NUR FUER URSPRUNGSVARIANTE DES IEC-TREIBERS */
/*---------------------------------------------*/

/* Eintrag im Datenmodul deva.. */
typedef struct {
	USINT	Nummer;
	USINT	Adresse;
	USINT	Aktiv;
	USINT	TimeSynch;
	UINT	AnlagenNr;
	UINT	Frei;
} DeviceType;

/* Eintrag im Datenmodul stoer.. */
typedef struct {
	USINT	Device;
	USINT	Type;
	USINT	F1;
	USINT	F2;
	UINT	Datentyp;
	UINT	DatenpunktNr;
} StoerDM_typ;

/* Eintrag im Datenmodul wert.. */
typedef struct {
	USINT	Device;
	USINT	Type;
	USINT	Info;
	USINT	WertCode;
	UINT	Datentyp;
	UINT	DatenpunktNr;
	UINT	Info1;
	UINT	Info2;
} WertType;

/* Struktur mruk */
typedef struct {
	USINT	Type;
	USINT	Info;
} MrukType;

/* Eintrag im Datenmodul norm */
typedef struct {
	INT		x1;
	INT		y1;
	INT		x2;
	INT		y2;
} NormierungType;

/*-------------------------------------------------------*/
/* BIS HIER: NUR FUER URSPRUNGSVARIANTE DES IEC-TREIBERS */
/*-------------------------------------------------------*/

/*--------------------------*/
/* NUR FUER VARIANTE DbSERV */
/*--------------------------*/

/* Struktur eines Datenpunkt Items im Speicher */
typedef struct {
	USINT	AccessCounter;					/* Zaehle fuer Zugriffe auf das Item */
	USINT	ErrorInfo;						/* Fehlerinformation */
	USINT	DeviceAdr;						/* Geraetadresse */
	USINT	KopplungsStoerung;				/* Item fuer Kopplungsstoerung*/
	USINT	TimeSynchError;					/* Item fuer Fehler bei Zeitsynchronisation: 0=undefiniert, 1= AUS (kein Fehler), 2= EIN (Fehler) */
	USINT	IECType;						/* IEC-Type */
	USINT	IECInfoNr;						/* IEC-Informations Nummer */
	USINT	IECAnalogNr;					/* IEC-Nummer des Analogwertes */
	USINT	MRuc;							/* MRuc verwenden 0=nein/1=ja */
	USINT	MRucType;						/* IEC-Type fuer MRuc */
	USINT	MRucInfo;						/* IEC-Informations Nummer fuer MRuc */
	USINT	Mode;							/* Mode fuer Digitalmeldungen */
	USINT	Normierung;						/* Normierung 0=nein / 1=ja */
	USINT	ItemTypNr;						/* Datentypnummer des Items */
	USINT	Invalid;						/* Invalid Bit des Analogwertes auswerten 0=nein 1=ja */
	USINT	Overflow;						/* Overflow Bit des Analogwertes auswerten 0=nein 1=ja */
	UINT	NormierungIdx;					/* Index fuer Normierung */
	UINT	DPNr;							/* Datenpunktnummer */
	UINT	DPTypNr;						/* Datentypnummer */
	UINT	ItemNr;							/* Item Nummer */
	DINT	ValueDevice;					/* Wert,der vom Geraet empfangen wurde */
	DINT	ValueServer;					/* Wert, der an den Server uebergeben wurde */
} IEC_DP_Info_typ;

/* Struktur eines Normierungseintrages im Speicher */
typedef struct {
	DINT	x1;								/* Eingangswert minimal */
	DINT	y1;								/* Ausgangswert minimal */
	DINT	x2;								/* Eingangswert maximal */
	DINT	y2;								/* Ausgangswert maximal */
} IEC_Normierung_typ;

/*------------------------------------*/
/* BIS HIER: NUR FUER VARIANTE DbSERV */
/*------------------------------------*/

/*-----------------------------------------------*/
/* Strukturen fuer die Verwaltung eines Geraetes */
/*-----------------------------------------------*/

/* Datentyp: Four Octet binary time */

typedef struct {
	USINT	MilliSeconds1;
	USINT	MilliSeconds2;
	USINT	Minutes;
	USINT	Hours;
} FourOctetBinaryTime_typ;

/* Datentyp: Seven Octet binary time */

typedef struct {
	USINT	MilliSeconds1;
	USINT	MilliSeconds2;
	USINT	Minutes;
	USINT	Hours;
	USINT	Day;
	USINT	Month;
	USINT	Year;
	USINT	not_used;
} SevenOctetBinaryTime_typ;

/* Information ueber die Uebertragung eines Stoerschriebes */
typedef struct {
	UINT						Number;						/* Nummer des Stoerschriebes (vom Geraet) */
	USINT						Status;						/* Status des Stoerschriebes (vom Geraet) */
	RTCtime_typ 				Time;						/* Zeitstempel des Stoerschriebes (vom Geraet) */
	SevenOctetBinaryTime_typ	IECTime;					/* Zeitstempel in IEC-Form */
	USINT						Clear;						/* Stoerschrieb kann geloescht werden */
	USINT						Transmitted;				/* Stoerschrieb wurde uebertragen */
	USINT						TypeOfValues;				/* Typ der zu übertragenden Daten */
} FaultInformationType;

/* Information ueber den Verbindungsstatus und den Telegrammverkehr */
typedef struct {
	USINT					Enabled;					/* Verbindung zum Geraet ist aktiviert */
	USINT					Adresse;					/* Geraeteadresse */
	USINT					Verbindungsversuche;
	USINT					ZeitsynchAktiv;
	USINT					StateTimeSynchError;
	UDINT					TimeoutTimeSynch;
	USINT					FCB_Toggle;
	USINT					KE_InitOk;
	UDINT					Timeout_KE;
	UINT					AdresseLeitsystem;
	UINT					AnlagenNr;
	UDINT					ZeitLetzteVerbindung;
	UDINT					ZeitLetzteZeitsync;
	USINT					Class1Request;
	USINT					TimoutNext;
	USINT					GI_Ok;
	UDINT					Timeout_GI;
	USINT					LetzterACD;
	UDINT					Class2Verz;
	USINT					Class1Verz;
	USINT					set_event;
	USINT					VerbindungsStoerung;
	UDINT					Timeouts;
	UDINT					VerbindungsStoerungen;
	UINT					LetzterVerbindungsfehler;
	USINT					NrOfFaults;					/* Anzahl vorhandener Stoerschriebe */
	USINT					FaultFunctionType;			/* Funktionsnummer */
	IEC_DP_Info_typ			*pFaultDPInfo;				/* Zeiger auf Datenpunkt-Info-Struktur im Speicher */
	FaultInformationType	FaultInfo[2];
	UINT					DPInfoFirstEntry;			/* Index des ersten Eintrages im Speicher fuer dieses Device */
	UINT					DPInfoLastEntry;			/* Index del letzten Eintrages im Speicher fuer dieses Device */
	DTStructure				TSynch;						/* Uhrzeit die zuletzt an das Geraet gesendet wurde */
	DTStructure				TDevice;					/* Uhrzeit die vom Geraet empfangen wurde */
	UDINT					TDiff;						/* Zeitdifferenz zwischen gesendeter und empfangener Uhrzeit */
	UINT					TDiffCounter;				/* Fehlerzaehler, Zeitdifferenz zu gross */
} DeviceActivType;

/* Struktur zur Verwaltung der Schnittstelle und des Sende- und Empfangsbuffers */
typedef struct {
	USINT					write_read_activ;
	UDINT					receive_timeout;
	UDINT					timeout;
	UDINT					Ident; 						/* pointer for ident info */
	USINT					WriteData[30];
	USINT					WriteDataLen;
	USINT					sendewiederholung;
	USINT					class1_res_adc1;
	USINT					ReadData[256]; 				/* arrays for write and read data */
	UDINT					RBufferAdr;
	UINT					OpenError;
	UINT					WriteErrorCount;			/* Zaehler fuer fehlerhafte Schreibversuche */
	UINT					WriteError;					/* Letzte Fehlernummer bei fehlerhaftem Schreibversuch */
	UINT					FirstWriteError;			/* Fehlernummer des ersten fehlerhaften Schreibversuches */
	UINT					LastWriteError;				/* Fehlernummer des letzten fehlerhaften Schreibversuches */
	UINT					ReOpenCount;				/* Zaehler, wieoft das Device neu geoeffnet wurde */
} ComType;

/* Struktur zur Verwaltung der verwendeten Datenmodule */
typedef struct{
	UDINT					AdrDM_stoer;
	UINT					MaxWerteDM_stoer;
	UDINT					AdrDM_wert;
	UINT					MaxWerteDM_wert;
	UDINT					AdrDM_mruk;
	UINT					MaxWerteDM_mruk;
	UDINT					AdrDM_norm;
	UINT					MaxWerteDM_norm;
} DMInfoType;

/* Struktur mit Infos ueber die verwendete Schnittstelle */
typedef struct {
	USINT 					StringDevice[32]; 			/* initialize strings for FRM_xopen */
	USINT 					StringMode[80]; 			/* initialize strings for FRM_xopen */
	FRM_xopen_typ			FrameXOpenStruct;
	XOPENCONFIG				XOpenConfigStruct;
} ComIniType;

/* Strukturen zur Uebertragung von Stoerschrieben */
/* Struktur des Headers fuer die Uebergabe an das Leitsystem */
typedef struct {
	UINT						FaultNumber;				/* Fehleridentifizierungsnummer */
	UINT						Status;
	SevenOctetBinaryTime_typ	FaultTime;					/* Zeitpunkt der Störung in IEC-Form */
	UINT						GridFaultNumber;			/* Netzstörungsnummer */
	USINT						NrOfStoredChannels;			/* Anzahl übertragener Kanäle */
	USINT						Res1;						/* Frei */
	UINT						NrOfElementsPerChannel; 	/* Anzahl Werte pro Kanal */
	UINT						IntervallTime;				/* Abtastzeit */
	FourOctetBinaryTime_typ		DistStartTime;				/* Startzeitpunkt der Aufzeichnung in IEC-Form */
	UINT						NrOfTags;					/* Anzahl übertragener Tags */
} DisturbanceHeadType;

/* Struktur eines Tags fuer die Uebergabe ans das Leitsystem */
typedef struct {
	UINT					DatenTyp;
	UINT					DatenpunktNr;
	UINT					Item;
	UINT					TagPosition;
	USINT					Value;
	USINT					Res1;
} DisturbanceTagType;

/* Struktur der Informationen (Teil 1) eines Kanales fuer die Uebergabe ans das Leitsystem */
typedef struct {
	UINT					DatenTyp;
	UINT					DatenpunktNr;
	UINT					Item;
} DisturbanceChannelInfoType;

/* Struktur der Informationen (Teil 2) eines Kanales fuer die Uebergabe ans das Leitsystem */
typedef struct {
	unsigned long			RPV;
	unsigned long			RSV;
	unsigned long			RFA;
} DisturbanceChannelFaktorType;

typedef struct {
	UINT					ErrorNr;					/* Letzte Fehluebertragung: Fehlerkennung */
	UINT					Function;					/* Letzte Fehluebertragung: Funktion */
	UINT					TypeOfOrder;				/* Letzte Fehluebertragung: Type of Order */
	UINT					ChannelNr;					/* Letzte Fehluebertragung: Kanalnummer */
}	DistTransErrorType;

/* Verwaltung der Uebertragung eines Stoerschriebes */
typedef struct {
	UINT					Function;					/* Momentane Übertragungsfunktion */
	USINT					DataSend;					/* Auftrag Daten senden */
	USINT					WaitForResponse;			/* Warten auf Antwort */
	USINT					TypeOfOrder;				/* Befehlskennung (abort, acknowledge,..) */
	USINT					DeviceAtWork;				/* Gerätenummer (1..) fuer Uebertragung (aus Array DeviceActiv) */
	USINT					FunctionType;				/* Funktionsnummer */
	USINT					TypeOfValues;				/* Typ der zu übertragenden Daten */
	UINT					NrOfReceivedTags;			/* Anzahl empfangener Tags */
	UINT					NrOfReceivedChannels;		/* Anzahl empfangender Kanäle */
	UINT					NrOfChannels;				/* Anzahl zu übertragender Kanäle */
	UINT					ActualChannelTyp;			/* Kennnummer des zu übertragenden Kanales */
	UINT					LastChannelTyp;				/* Kennnummer des zuletzt uebertragenen Kanales */
	UINT					EstimateChannelPos;			/* Erwartete Startposition */
	USINT					NewChannel;					/* Ein neuer Kanal wird uebertragen */
	USINT					StoreChannel;				/* Analogkanal speichern */
	UINT					ChannelDataError;			/* Fehlermerker, falls beim Uebertragen eines Kanales Fehler auftreten */
	UDINT					TimeOut;					/* Timeoutzaehler */
	USINT					Trys;						/* Versuche Daten zu uebertragen */
	USINT					FaultIdx;					/* Index zu uebertragenden Stoerschriebes */
	USINT					BufferIdx;					/* Bufferindex fuer die Stoerschriebdaten */
	UINT					Delay;						/* Verzoegerung beim Empfangen von Stoerschrieben gleicher Stationen */
	DistTransErrorType		ActError;					/* Fehlerspeicher fuer laufende Uebertragung */
	DistTransErrorType		LastError;					/* Fehlerspeicher der letzten Uebertragung */
} DisturbanceDataType;

/* Struktur zur Ausloesung von Kommandos */
typedef struct {
	UINT					Function;					/* Momentane Übertragungsfunktion */
	USINT					DataSend;					/* Auftrag Daten senden */
	USINT					WaitForResponse;			/* Warten auf Antwort */
	USINT					DeviceAdress;				/* GeräteAdresse (alternativ DeviceAtWork) */
	USINT					DeviceAtWork;				/* Gerätenummer (alternativ DeviceAdress) (1..) fuer Uebertragung (aus Array DeviceActiv) */
	USINT					FunctionType;				/* Funktionsnummer */
	USINT					InformationNumber;			/* Informationsnummer */
	USINT					Val;						/* Wert, der zu schreiben ist */
	USINT					ReturnVal;					/* Wert, der vom Geraet zurueckgemeldet wurde */
	USINT					ReturnInformation;			/* Rueckmeldungswert */
	UINT					TimeOut;					/* Timeoutzaehler */
	USINT					Trys;						/* Versuche Daten zu uebertragen */
	USINT					Ready;						/* Kommando uebertragen */
	UINT					Error;						/* Fehlermeldung */
} CommandType;

/* Struktur zur Vewaltung einer gesamten Linie */
typedef struct {

	UINT					LinienNummer;
	UINT					SNr;
	DeviceType 				DeviceTAB[DEVICES_PRO_LINE];
	DeviceActivType 		DeviceActiv[DEVICES_PRO_LINE];
	DisturbanceDataType		DistData;
	DisturbanceHeadType		DistHead;
	CommandType				Command;
	USINT 					DeviceAtWork;
	USINT					Error;
	USINT					ComStart;
	DMInfoType				dm;
	ComType					com;
} AnlagenType;

/* Struktur zum Speichern von Kontrollelementen der Telegramme */

typedef struct {
	USINT				ACD;
	USINT				DFC;
	USINT				Function;
} ControlFieldPrimary_typ;

/* Strukturen fuer Testzwecke */
typedef struct {
	USINT 					enable;
	USINT					ready;
	UINT					LinienNummer;
	USINT 					DeviceAdresse;
	USINT 					FunctionType;
	USINT 					InformationNumber;
	USINT 					Messwert;
} TestTypeDig;

typedef struct {
	USINT 					enable;
	USINT					ready;
	UINT					LinienNummer;
	USINT 					DeviceAdresse;
	USINT 					FunctionType;
	USINT 					InformationNumber;
	USINT 					AnzahlMesswerte;
	INT 					Messwerte[MAX_ANALOGWERTE];
} TestTypeAna;

typedef struct {
	USINT 					enable;
	USINT 					Adresse;
} TestTypeGlobal;

typedef struct {
	USINT					DataReady;
	USINT					ClearData;
	USINT					BufferIdx;
} DisturbanceDataServer;

typedef struct {
	USINT					Code;
	USINT					SetEventStream;
	DeviceActivType			*DevicePointer;
	UINT					FaultNumber;
	UDINT					DataLen;
	UDINT					DataAdr;
	UDINT					Size;
	UINT					status;
} DisturbanceBufferInfo;

typedef struct {
	UINT					NrOfBuffers;
	DisturbanceBufferInfo	Info[NR_OF_BUFFERS];
} DisturbanceBuffer;

typedef union
{
	BOOL 	b;
	SINT 	i1;
	USINT	ui1;
	INT		i2;
	UINT	ui2;
	DINT	i4;
	UDINT	ui4;
	float r4;
} PAR_TYPE;

/**********************************************************
*						Prototypen
**********************************************************/
void Zeitmessung(AnlagenType *pANL);

void Device_Reaktivieren(AnlagenType *pANL);

USINT Data_write(AnlagenType *pANL);

void Data_read(AnlagenType *pANL);

USINT save_analogwert(	DMInfoType *pDMInfo, UINT LinienNummer, DeviceActivType *pDeviceActiv,
						USINT FunctionType, USINT InformationNumber, USINT AnzahlMesswerte,
						USINT *AdresseMesswerte, USINT set_event);

USINT save_analogwert_priv(	DMInfoType *pDMInfo, UINT LinienNummer, DeviceActivType *pDeviceActiv,
							USINT FunctionType, USINT InformationNumber, USINT AnzahlMesswerte,
							USINT *AdresseMesswerte, USINT set_event);

USINT save_counter_2(DMInfoType *pDMInfo, UINT LinienNummer, DeviceActivType *pDeviceActiv,
							USINT FunctionType, USINT InformationNumber, USINT AnzahlMesswerte,
							USINT *AdresseMesswerte, USINT set_event);

void save_analogwert_error(	DMInfoType *pDMInfo, UINT LinienNummer, DeviceActivType *pDeviceActiv,
						USINT FunctionType,USINT InformationNumber, USINT set_event);

USINT save_digitalwert( DMInfoType *pDMInfo, UINT LinienNummer, DeviceActivType *pDeviceActiv,
						USINT FunctionType,USINT InformationNumber, USINT Messwert,
						RTCtime_typ *TimeBuf, USINT set_event);

USINT save_kopplungsstoerung( DMInfoType *pDMInfo, UINT LinienNummer, DeviceActivType *pDeviceActiv, USINT Messwert, RTCtime_typ *TimeBuf, USINT set_event);

USINT save_TimeSynchError( DMInfoType *pDMInfo, UINT LinienNummer, DeviceActivType *pDeviceActiv, USINT Messwert, RTCtime_typ *TimeBuf, USINT set_event);

void get_4OctetBinaryTime(USINT *data, RTCtime_typ *TimeBuf, RTCtime_typ *SysTime);

void get_7OctetBinaryTime(USINT *data, RTCtime_typ *TimeBuf, RTCtime_typ *SysTime);

void debug_initialize(void);

void debug_open_device(USINT enable);

short int send_buffer(ComType *pCom, UINT LinienNummer, USINT Adresse);

void clear_buffer(ComType *pCom);

USINT MakeCRC(char *data, USINT start, USINT laenge);

void Reset_KE(UINT LinienNummer, DeviceActivType *pDeviceActiv, ComType *pCom);

void Zeit_Sync(UINT LinienNummer,DeviceActivType *pDeviceActiv, ComType *pCom);

void Init_GI(UINT LinienNummer,DeviceActivType *pDeviceActiv, ComType *pCom);

void Class_1_Request(UINT LinienNummer,DeviceActivType *pDeviceActiv, ComType *pCom);

void Class_2_Request(UINT LinienNummer,DeviceActivType *pDeviceActiv, ComType *pCom);

void disturbance_data_request(AnlagenType *pANL);

void disturbance_data_response(AnlagenType *pANL,USINT code, USINT info);

void disturbance_data_timeout(AnlagenType *pANL);

void clear_dist_data_request(AnlagenType *pANL);

signed short save_disturbance_data(UINT code, AnlagenType *pANL);

void check_device_dist_data(AnlagenType *pANL);

void check_dist_data_transmission();

void abort_disturbance_data(AnlagenType *pANL);

void save_disturbance_error(AnlagenType *pANL,UINT Error, UINT Function, UINT TypeOfOrder, UINT Channel);

void command_request(AnlagenType *pANL);

void command_timeout(AnlagenType *pANL);

void command_response(AnlagenType *pANL);

void GetNewDevice(AnlagenType *pANL);

void Empfangsfehler(UINT nr, AnlagenType *pANL);

void timesynch_timeout(AnlagenType *pANL);

USINT check_m1(AnlagenType *pANL);

USINT check_m2(AnlagenType *pANL);

USINT check_m3(AnlagenType *pANL);

USINT check_m5(AnlagenType *pANL);

USINT check_m6(AnlagenType *pANL);

USINT check_m8(AnlagenType *pANL);

USINT check_m9(AnlagenType *pANL);

USINT check_m23(AnlagenType *pANL);

USINT check_m26(AnlagenType *pANL);

USINT check_m27(AnlagenType *pANL);

USINT check_m28(AnlagenType *pANL);

USINT check_m29(AnlagenType *pANL);

USINT check_m30(AnlagenType *pANL);

USINT check_m31(AnlagenType *pANL);

USINT check_m79(AnlagenType *pANL);

USINT check_m205(AnlagenType *pANL);

void tel_ok(AnlagenType *pANL);

void get_idBrServer();

void disturbance_simulation();

BOOL DeviceIsActive(AnlagenType *pANL, USINT DeviceAddr);

/**********************************************************
*				Globale Variablen Declaration
**********************************************************/

/**********************************************************
*				Lokale Variablen Declaration
**********************************************************/

_LOCAL	IEC_Config_typ					IEC_Config;

_LOCAL	UDINT							myidBrServer;
_LOCAL_RETAIN	UINT							statePV_xgetadr;
_LOCAL	UDINT							pv_adresse, data_len;
_LOCAL  UINT							StatusSetValueItem;
_LOCAL	UINT							SetEventStreamStatus;
_LOCAL	UINT							RelEventStreamStatus;

_LOCAL	RTInfo_typ						rt_info;
_LOCAL  UINT							CycleTime;

_LOCAL AnlagenType						stANL[MAX_LINES];
_LOCAL  ComIniType						stComIni[MAX_LINES];
_LOCAL RTCtime_typ						RPSTime;
_LOCAL USINT							RPSTimeOK;

_LOCAL DisturbanceDataServer			DistDataServer;
_LOCAL UINT								DistDataType;
_LOCAL UINT								DistDataPoint;

_LOCAL FRM_rbuf_typ						FrameReleaseBufferStruct;
_LOCAL FRM_close_typ 					FrameCloseStruct;
_LOCAL FRM_write_typ					FrameWriteStruct;
_LOCAL FRM_read_typ						FrameReadStruct;
_LOCAL FRM_write_typ					DebugWriteStruct;

_LOCAL RTCtime_typ 						TimeBuf;

_LOCAL USINT 							Error,ReadError;
_LOCAL UINT								StatusRead, StatusReleaseBuffer;
_LOCAL UDINT 							*ReadBuffer; 								/* pointer to read buffer */
_LOCAL UINT  							*ReadBufferLen;
_LOCAL UINT 							ReadBufferLength;

_LOCAL UINT								EFehler;
_LOCAL USINT							EmpfangeneMesswerte,InfoElemente;

_LOCAL	DatObjInfo_typ					DOI_wert[MAX_LINES],DOI_deva[MAX_LINES],DOI_stoer[MAX_LINES],DOI_mruk,DOI_norm,DOI_lines;
_LOCAL	DatObjRead_typ					DOR_wert[MAX_LINES],DOR_deva[MAX_LINES],DOR_stoer[MAX_LINES],DOR_mruk,DOR_norm,DOR_lines;

_LOCAL	DisturbanceTagType				DisturbanceTagInfo;
_LOCAL	DisturbanceChannelInfoType		DisturbanceChannelInfo;
_LOCAL	DisturbanceChannelFaktorType	DisturbanceChannelFaktor;

_LOCAL	unsigned long					ChannelDataLen,CopySize,Offset,Anzahl,Adresse;
_LOCAL	unsigned short					StartNr;
_LOCAL	USINT							FunctionType,InformationNumber,NrOfTags,aktTag;
_LOCAL	USINT							Messwert,WertLS0,WertLS1,found;

_LOCAL	DisturbanceBuffer				DataBuffer;

_LOCAL UINT								ActiveLines;
_LOCAL USINT							aktANL,maxANL;

_LOCAL ControlFieldPrimary_typ			ControlFieldPrimary;

_LOCAL TestTypeDig						DigTest;
_LOCAL TestTypeAna						AnaTest;
_LOCAL TestTypeGlobal					GlobalTest;

_LOCAL	DatObjInfo_typ					DOISimu;
_LOCAL	BOOL							DisturbanceSimulation;

_LOCAL_RETAIN Stats_Typ						SYS_Statistic	;

_LOCAL	USINT							Overflow[MAX_ANALOGWERTE];
_LOCAL	USINT							Invalid[MAX_ANALOGWERTE];

_LOCAL USINT IEC_Info_Clear;
_LOCAL USINT IEC_Info_Enable;

/*** eof *****************************************************************************/
```
